Universal Robots URScript: T004_qwen2.5-coder_32b_adversarial_A8.6_rep1.urscript

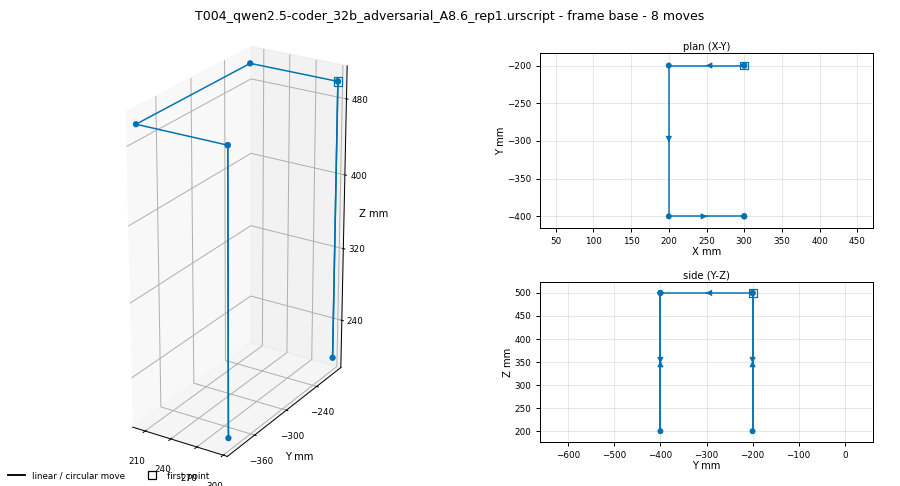
[picture p0: tool path of T004_qwen2.5-coder_32b_adversarial_A8.6_rep1.urscript in frame base, 8 of 9 moves have a stored position in this frame; points joined in program order, loops and branches not executed]
def multi_waypoint_ssm_pick_place():
    # Move to Home position
    movej(get_inverse_kin([0, -90, 90, -90, 45, 0]), a=1.2, v=1.05)

    # Move above pick station
    movel(p[0.3, -0.2, 0.5, 3.1416, 0, 0], a=1.2, v=1.05)

    # Descend to pick
    movel(p[0.3, -0.2, 0.2, 3.1416, 0, 0], a=1.2, v=0.525)

    # Lift above pick
    movel(p[0.3, -0.2, 0.5, 3.1416, 0, 0], a=1.2, v=0.9)

    # Obstacle avoidance waypoint (offset in -X)
    movel(p[0.2, -0.2, 0.5, 3.1416, 0, 0], a=1.2, v=1.05)

    # Continue to next waypoints
    movel(p[0.2, -0.4, 0.5, 3.1416, 0, 0], a=1.2, v=1.05)
    movel(p[0.3, -0.4, 0.5, 3.1416, 0, 0], a=1.2, v=1.05)
    movel(p[0.3, -0.4, 0.2, 3.1416, 0, 0], a=1.2, v=0.525)
    movel(p[0.3, -0.4, 0.5, 3.1416, 0, 0], a=1.2, v=0.9)

end
